FUNCTION_BLOCK WagoSystemWithIO (* Composite Function Block Type *)
  (* Standard: 61499-2 *)
  (* Version 0.2, 2003-12-05, JHC, Rockwell Automation, Renamed from NEWCOMPFB. *)
  (* Compiler header: package fb.rt.wago; *)
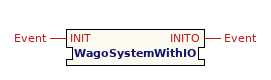
  EVENT_INPUT
    INIT; (* Initialization Request *)
  END_EVENT
  EVENT_OUTPUT
    INITO; (* Initialization Confirm *)
  END_EVENT
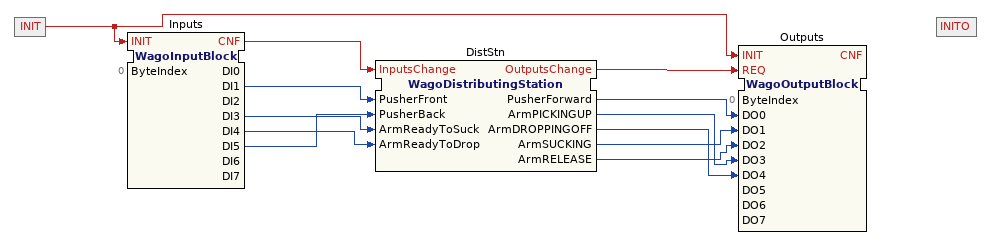
  FBS
    DistStn : WagoDistributingStation;
    Inputs : WagoInputBlock(ByteIndex := 0);
    Outputs : WagoOutputBlock(ByteIndex := 0);
  END_FBS
  EVENT_CONNECTIONS
    INIT TO Inputs.INIT;
    INIT TO Outputs.INIT;
    Inputs.CNF TO DistStn.InputsChange;
    DistStn.OutputsChange TO Outputs.REQ;
  END_CONNECTIONS
  DATA_CONNECTIONS
    Inputs.DI1 TO DistStn.PusherFront;
    Inputs.DI5 TO DistStn.PusherBack;
    Inputs.DI3 TO DistStn.ArmReadyToSuck;
    Inputs.DI4 TO DistStn.ArmReadyToDrop;
    DistStn.PusherForward TO Outputs.DO0;
    DistStn.ArmPICKINGUP TO Outputs.DO3;
    DistStn.ArmDROPPINGOFF TO Outputs.DO4;
    DistStn.ArmSUCKING TO Outputs.DO1;
    DistStn.ArmRELEASE TO Outputs.DO2;
  END_CONNECTIONS
END_FUNCTION_BLOCK
